FUNCTION_BLOCK FB_ValveBank IMPLEMENTS I_ValveBank
VAR_INPUT
    nNumOfValves 	: INT;		// Total number of valves in this bank
	nValveMaskAuto 	: DWORD;	// Each bit enables corresponding valve 
END_VAR
VAR_IN_OUT
    afbValve 		: ARRAY[0..nNumOfValves - 1] OF FB_Valve; // Max size; NumOfValves limits how many are used
	anReqOpenManual	: ARRAY[0..nNumOfValves - 1] OF BOOL; 
	anReqCloseManual: ARRAY[0..nNumOfValves - 1] OF BOOL;
END_VAR
VAR_OUTPUT
    aeValveStatus : ARRAY[0..nNumOfValves -1] OF E_ValveStatus;
    bHasAnyError : BOOL;
END_VAR

METHOD M_Status
VAR
    i : INT;
END_VAR
bHasAnyError := FALSE;
FOR i := 0 TO nNumOfValves - 1 DO

	aeValveStatus[i] := afbValve[i].M_Status();
	
	IF aeValveStatus[i] <> OK THEN
		bHasAnyError := TRUE;
    END_IF
	
END_FOR


//OR mapp the VB Status  bits here
END_METHOD

METHOD M_TriggerFromMask : BOOL
VAR
    i : INT;
    bitSet : BOOL;
END_VAR

FOR i := 0 TO nNumOfValves - 1 DO
    bitSet := (nValveMaskAuto AND SHL(1, i)) <> 0;
    
    IF aeValveStatus[i] = OK THEN
        IF bitSet THEN
            afbValve[i].M_Open();
        ELSE
            afbValve[i].M_Close();
        END_IF
    END_IF
END_FOR

M_TriggerFromMask := TRUE;
END_METHOD

METHOD M_TriggerManual
VAR
    i : INT;
END_VAR
FOR i := 0 TO nNumOfValves - 1 DO
    IF NOT aValveError[i] THEN
        
		IF anReqOpenManual[i] THEN
			afbValve[i].M_Open(); 
		ELSE	
			afbValve[i].M_Close(); 
		END_IF
		
    END_IF
END_FOR
END_METHOD

END_FUNCTION_BLOCK

(* stored: Version 1.1.0.1, ProductVersion 3.1.4024.15
   POU FB_ValveBank: Id {6fd479d4-9175-4488-b2ec-fe7d4059738b}, SpecialFunc None
   Method M_Status: Id {49dfdca5-5b79-4752-a62e-fc568e236d58}
   Method M_TriggerFromMask: Id {fe376a1d-db65-4f96-89c4-385f8cf1d130}
   Method M_TriggerManual: Id {8af14a3c-2dc8-4674-a94b-adeb0c9e665c} *)
